PROGRAM prgPerf
VAR
	hugeArrayOfComplex : stHugeArrayOfComplex;
	hugeArrayOfPrimitive : stHugeArrayOfPrimitive;
	hugeStructureOfComplex : stHugeStructureOfComplex;	
	hugeStructureOfPrimitive : stHugeStructureOfPrimitive;	
END_VAR

END_PROGRAM

(* stored: Version 1.1.0.1, ProductVersion 3.1.4024.6
   POU prgPerf: Id {cacd3814-60ec-466a-91b2-73a55b6b21a8}, SpecialFunc None *)
